(*
SPDX-FileCopyrightText: © 2026 Oleksandr Tiutyk <trofimich@gmail.com>
SPDX-License-Identifier: MIT
License: https://opensource.org/license/mit
*)

(*!
<summary>
Beckhoff EL1018_EX: Extended 8-channel fast digital input terminal with diagnostics.
</summary>
<description>
Extends EL1018 with EtherCAT Working Counter and slave state diagnostics.
When used for I/O, link located fields or their containing buffers to the matching selected PDOs.
The record is not a packed wire buffer; compiler padding is not part of the device specification.
Unlinked/default values do not prove valid I/O. The caller evaluates bus/channel validity before use.
Use one owner task per instance and externally synchronize other access; multi-field snapshots are not atomic.
Copies store data without creating hardware links. Keep borrowed field references valid while consumers are bound.
This passive record performs no validation, synchronization, configuration or protocol advancement.
WcState=TRUE means process-data exchange is invalid. State is acyclic EtherCAT/link information,
not proof of current measurement validity. Link diagnostics to the matching slave InfoData entries.
The selected PDO representation is documented by the base terminal model.
InputToggle signals an input update by changing state; TRUE alone does not mean fresh data.
</description>
*)
TYPE EL1018_EX EXTENDS EL1018:
STRUCT
	WcState AT %I* : BOOL;
	InputToggle AT %I* : BOOL;
	State AT %I* : UINT;
END_STRUCT
END_TYPE

(* stored: Version 1.1.0.1, ProductVersion 3.1.4026.18
   DUT EL1018_EX: Id {f1fb739d-5028-491a-890c-d0561d16145b} *)
